(* IEC 61131-3 sources: plc_generation_empirical_study/datasets_100/tasks/C04_S17_lean_composite, 2 files *)

(* ---- interface.st ---- *)
FUNCTION_BLOCK C04_S17_lean_composite
VAR_INPUT
    A_AutoMode : BOOL;
    A_AutoDemand : BOOL;
    A_ManualDemand : BOOL;
    A_SafetyOK : BOOL;
    A_Inhibit : BOOL;
    B_EventA : BOOL;
    B_EventB : BOOL;
    B_Arm : BOOL;
    B_Reset : BOOL;
    SubsystemBEnable : BOOL;
    CrossReset : BOOL;
END_VAR
VAR_OUTPUT
    A_Command : BOOL;
    A_Blocked : BOOL;
    B_Captured : BOOL;
    B_Code : INT;
    B_Pulse : BOOL;
    CrossReady : BOOL;
    CrossBlocked : BOOL;
END_VAR
END_FUNCTION_BLOCK

(* ---- reference.st ---- *)
FUNCTION_BLOCK C04_S17_lean_composite
VAR_INPUT
    A_AutoMode : BOOL;
    A_AutoDemand : BOOL;
    A_ManualDemand : BOOL;
    A_SafetyOK : BOOL;
    A_Inhibit : BOOL;
    B_EventA : BOOL;
    B_EventB : BOOL;
    B_Arm : BOOL;
    B_Reset : BOOL;
    SubsystemBEnable : BOOL;
    CrossReset : BOOL;
END_VAR
VAR_OUTPUT
    A_Command : BOOL;
    A_Blocked : BOOL;
    B_Captured : BOOL;
    B_Code : INT;
    B_Pulse : BOOL;
    CrossReady : BOOL;
    CrossBlocked : BOOL;
END_VAR
VAR
    B_PrevA : BOOL := FALSE;
    B_PrevB : BOOL := FALSE;
END_VAR

A_Command := ((A_AutoMode AND A_AutoDemand) OR ((NOT A_AutoMode) AND A_ManualDemand))
           AND A_SafetyOK AND (NOT A_Inhibit);
A_Blocked := ((A_AutoMode AND A_AutoDemand) OR ((NOT A_AutoMode) AND A_ManualDemand))
           AND ((NOT A_SafetyOK) OR A_Inhibit);

IF CrossReset THEN
    CrossReady := FALSE;
ELSIF A_Command THEN
    CrossReady := TRUE;
END_IF;
CrossBlocked := SubsystemBEnable AND (NOT CrossReady);

IF SubsystemBEnable AND CrossReady THEN
    B_Pulse := FALSE;
    IF B_Reset THEN
        B_Captured := FALSE;
        B_Code := 0;
    ELSIF B_Arm AND (NOT B_Captured) THEN
        IF B_EventA AND (NOT B_PrevA) THEN
            B_Captured := TRUE;
            B_Code := 1;
            B_Pulse := TRUE;
        ELSIF B_EventB AND (NOT B_PrevB) THEN
            B_Captured := TRUE;
            B_Code := 2;
            B_Pulse := TRUE;
        END_IF;
    END_IF;
    B_PrevA := B_EventA;
    B_PrevB := B_EventB;
ELSE
    B_Captured := FALSE;
    B_Code := 0;
    B_Pulse := FALSE;
END_IF;

END_FUNCTION_BLOCK
